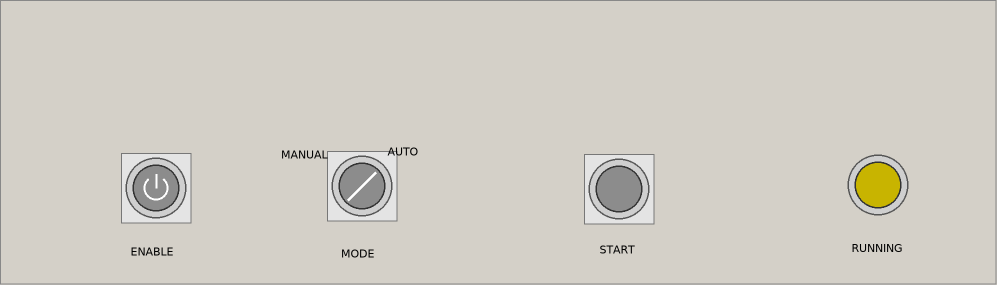
VISUALIZATION CraneHMI  // 997x285
    Lamp1 (843,150 70x70), style: Lamp-Lamp1-Yellow
    PowerSwitch (121,153 70x70), behaviour: TOGGLE, style: Switch-PowerSwitch-Gray
    RotarySwitch (327,151 70x70), behaviour: TOGGLE, style: Switch-RotarySwitch-Gray
    PushSwitch (584,154 70x70), behaviour: TOGGLE, style: Switch-PushSwitch-Gray
    Label (757,220 240x57), "RUNNING"
    Label (224,223 268x62), "MODE"
    Label (77,237 150x30), "ENABLE"
    Label (542,235 150x30), "START"
    Label (252,136 105x38), "MANUAL"
    Label (315,120 176x64), "AUTO"
END_VISUALIZATION

(* stored: Version 1.1.0.1, ProductVersion 3.1.4024.10
   Visu CraneHMI: Id {37617518-84c7-4410-8fbe-937cd6396db3} *)
